(* IEC 61131-3 sources: CodesysTest/export/SX_1195.dev/Plc Logic/Application/PRJ Specific/Motion/Motors/Applied Motion/Applied Motion TSM34IP-3DG/FB_SlaveAppliedMotionMotorEIP.pou, 2 files *)

(* ---- FB_SlaveAppliedMotionMotorEIP.pou.st ---- *)
(*#-#-#-#-#-#-#-#-#-#---Declaration---#-#-#-#-#-#-#-#-#-#-#-#-#*)

FUNCTION_BLOCK FB_SlaveAppliedMotionMotorEIP EXTENDS FB_BaseAppliedMotionMotorEIP
VAR_INPUT
	tensionFault : BOOL;
	torque : REAL;
END_VAR
VAR
	commsFailureONS : FB_ONS;
END_VAR
(*#-#-#-#-#-#-#-#-#-#---Implementation---#-#-#-#-#-#-#-#-#-#-#-#-#*)

//	Function Block: FB_SlaveAppliedMotionMotorEIP()
//	Description: A PLCOpen Motion compliant library for a Oriental AZ Series drive/motor
//	Created by: Evan Ische
//	Created Date: Tuesday, October 13th 2020

// Outputs for Motion Lib
operational := PowerOn;
EnableState := DriveEnable;

// Exit if drive isn't enabled.
IF NOT DriveEnable THEN
	error := FALSE;
	RETURN;
END_IF

SUPER^();

commsFailureONS(CLK := commsFailure);
IF commsFailureONS.OSF THEN
	THIS^.SetTorqueValue(THIS^.torque);
END_IF

(* ---- SetTorqueValue.m.st ---- *)
(*#-#-#-#-#-#-#-#-#-#---Declaration---#-#-#-#-#-#-#-#-#-#-#-#-#*)

METHOD SetTorqueValue : BOOL
VAR_INPUT
	torque : REAL;
END_VAR
VAR CONSTANT
	UPDATE_TORQUE_CMD : DINT := 16#4743;
END_VAR
(*#-#-#-#-#-#-#-#-#-#---Implementation---#-#-#-#-#-#-#-#-#-#-#-#-#*)

_sclCommand := UPDATE_TORQUE_CMD;
_parameter1 := TO_DINT(torque * 100);
_commands.SendHostCommand := TRUE;
